Staubli VAL3: onF4Event.pgx

program onF4Event()
  local num i
  local string l_sMessage
  local string l_sPage
  local string l_sItem
begin
  // look if the bButton is enable
  if bButton[3]
    l_sPage="Disk://goHome/page_home_set"
    call loadPage(l_sPage,l_sItem)
    logMsg("Disk://goHome/page_home_set")
  endIf
end
